// TIA Portal V19 export
FUNCTION "GreiderStyring" : Void   // FC2, LAD
{ S7_Optimized_Access := 'TRUE' }
// stored: SetENOAutomatically false
   VAR_TEMP   // added for the SCL form of the ladder/FBD networks
      _w1 : Bool;
   END_VAR
BEGIN

REGION Network 1
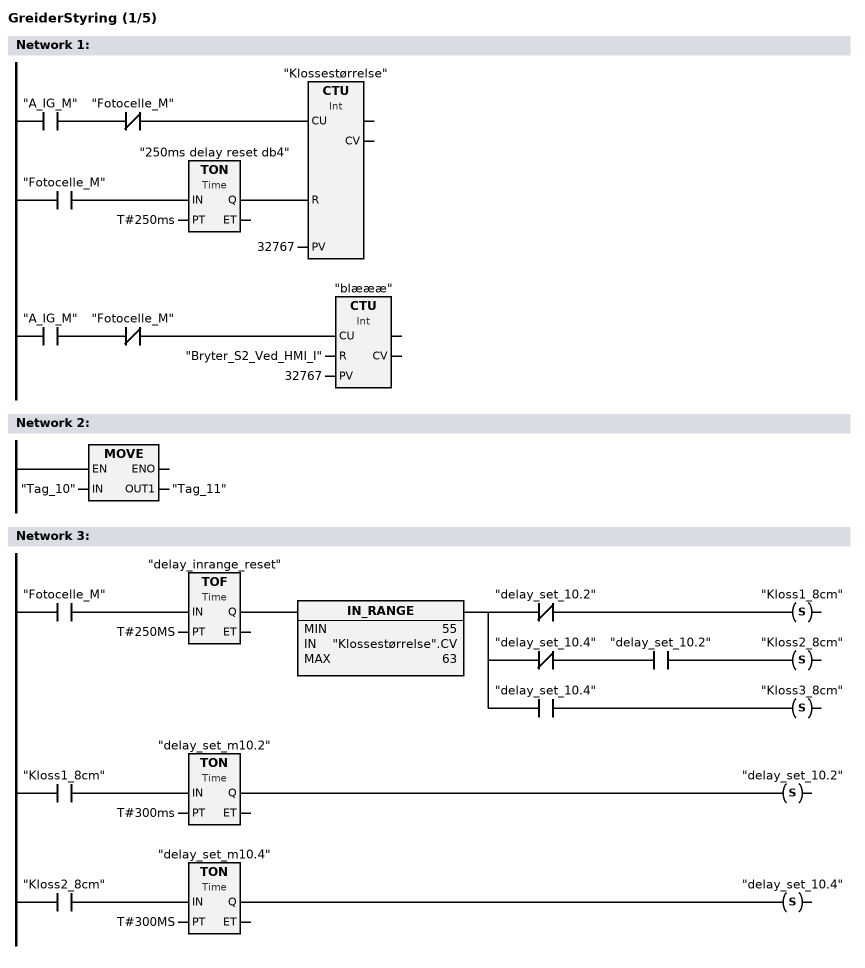
   RUNG wire#powerrail
      Contact( "A_IG_M" )
      I_Contact( "Fotocelle_M" )
      { S7_Templates := "value_type := Int" } "Klossestørrelse".CTU(r := wire#w1, pv := 32767, cv =>)
   END_RUNG
   RUNG wire#powerrail
      Contact( "Fotocelle_M" )
      { S7_Templates := "time_type := Time" } "250ms delay reset db4".TON(pt := T#250ms, et =>)
   END_RUNG wire#w1
   RUNG wire#powerrail
      Contact( "A_IG_M" )
      I_Contact( "Fotocelle_M" )
      { S7_Templates := "value_type := Int" } "blæææ".CTU(r := "Bryter_S2_Ved_HMI_I", pv := 32767, cv =>)
   END_RUNG
   // the same network as SCL:
   "250ms delay reset db4".TON(IN := "Fotocelle_M", PT := T#250ms);
   "Klossestørrelse".CTU(CU := "A_IG_M" AND NOT "Fotocelle_M", R := "250ms delay reset db4".Q, PV := 32767);
   "blæææ".CTU(CU := "A_IG_M" AND NOT "Fotocelle_M", R := "Bryter_S2_Ved_HMI_I", PV := 32767);
END_REGION

REGION Network 2
   RUNG wire#powerrail
      Move(in := "Tag_10", out1 => "Tag_11")
   END_RUNG
   // the same network as SCL:
   "Tag_11" := "Tag_10";
END_REGION

REGION Network 3
   RUNG wire#powerrail
      Contact( "Fotocelle_M" )
      { S7_Templates := "time_type := Time" } "delay_inrange_reset".TOF(pt := T#250MS, et =>)
      { S7_Templates := "SrcType := Int" } InRange(min := 55, in := "Klossestørrelse".CV, max := 63)
      wire#w1
      I_Contact( "delay_set_10.2" )
      S_Coil( "Kloss1_8cm" )
   END_RUNG
   RUNG wire#w1
      I_Contact( "delay_set_10.4" )
      Contact( "delay_set_10.2" )
      S_Coil( "Kloss2_8cm" )
   END_RUNG
   RUNG wire#w1
      Contact( "delay_set_10.4" )
      S_Coil( "Kloss3_8cm" )
   END_RUNG
   RUNG wire#powerrail
      Contact( "Kloss1_8cm" )
      { S7_Templates := "time_type := Time" } "delay_set_m10.2".TON(pt := T#300ms, et =>)
      S_Coil( "delay_set_10.2" )
   END_RUNG
   RUNG wire#powerrail
      Contact( "Kloss2_8cm" )
      { S7_Templates := "time_type := Time" } "delay_set_m10.4".TON(pt := T#300MS, et =>)
      S_Coil( "delay_set_10.4" )
   END_RUNG
   // the same network as SCL:
   "delay_inrange_reset".TOF(IN := "Fotocelle_M", PT := T#250MS);
   #_w1 := "delay_inrange_reset".Q AND (55 <= "Klossestørrelse".CV) AND ("Klossestørrelse".CV <= 63);
   IF #_w1 AND NOT "delay_set_10.2" THEN "Kloss1_8cm" := TRUE; END_IF;
   IF #_w1 AND NOT "delay_set_10.4" AND "delay_set_10.2" THEN "Kloss2_8cm" := TRUE; END_IF;
   IF #_w1 AND "delay_set_10.4" THEN "Kloss3_8cm" := TRUE; END_IF;
   "delay_set_m10.2".TON(IN := "Kloss1_8cm", PT := T#300ms);
   IF "delay_set_m10.2".Q THEN "delay_set_10.2" := TRUE; END_IF;
   "delay_set_m10.4".TON(IN := "Kloss2_8cm", PT := T#300MS);
   IF "delay_set_m10.4".Q THEN "delay_set_10.4" := TRUE; END_IF;
END_REGION

REGION Network 4
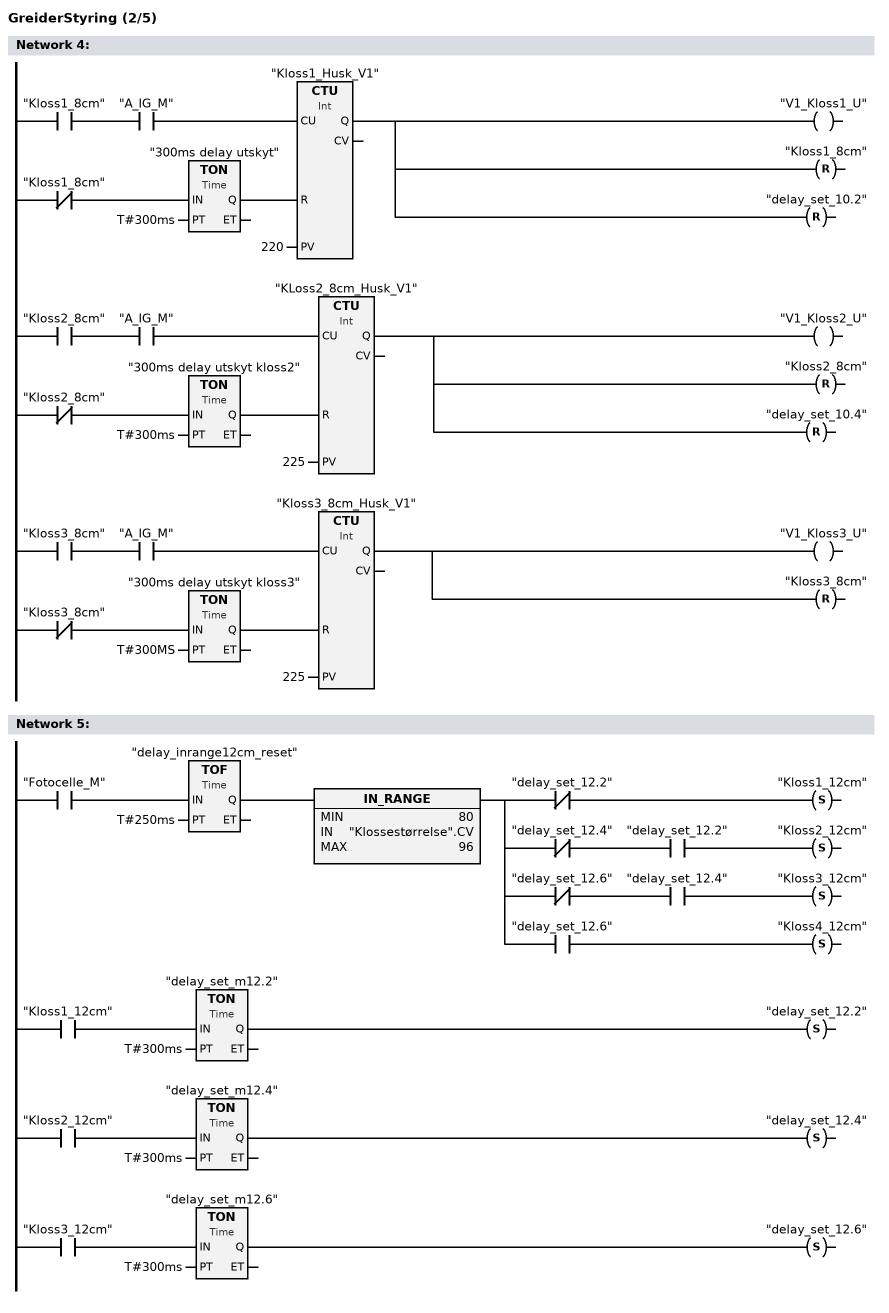
   RUNG wire#powerrail
      Contact( "Kloss1_8cm" )
      Contact( "A_IG_M" )
      { S7_Templates := "value_type := Int" } "Kloss1_Husk_V1".CTU(r := wire#w1, pv := 220, cv =>)
      wire#w2
      Coil( "V1_Kloss1_U" )
   END_RUNG
   RUNG wire#powerrail
      I_Contact( "Kloss1_8cm" )
      { S7_Templates := "time_type := Time" } "300ms delay utskyt".TON(pt := T#300ms, et =>)
   END_RUNG wire#w1
   RUNG wire#w2
      R_Coil( "Kloss1_8cm" )
   END_RUNG
   RUNG wire#w2
      R_Coil( "delay_set_10.2" )
   END_RUNG
   RUNG wire#powerrail
      Contact( "Kloss2_8cm" )
      Contact( "A_IG_M" )
      { S7_Templates := "value_type := Int" } "KLoss2_8cm_Husk_V1".CTU(r := wire#w3, pv := 225, cv =>)
      wire#w4
      Coil( "V1_Kloss2_U" )
   END_RUNG
   RUNG wire#powerrail
      I_Contact( "Kloss2_8cm" )
      { S7_Templates := "time_type := Time" } "300ms delay utskyt kloss2".TON(pt := T#300ms, et =>)
   END_RUNG wire#w3
   RUNG wire#w4
      R_Coil( "Kloss2_8cm" )
   END_RUNG
   RUNG wire#w4
      R_Coil( "delay_set_10.4" )
   END_RUNG
   RUNG wire#powerrail
      Contact( "Kloss3_8cm" )
      Contact( "A_IG_M" )
      { S7_Templates := "value_type := Int" } "Kloss3_8cm_Husk_V1".CTU(r := wire#w5, pv := 225, cv =>)
      wire#w6
      Coil( "V1_Kloss3_U" )
   END_RUNG
   RUNG wire#powerrail
      I_Contact( "Kloss3_8cm" )
      { S7_Templates := "time_type := Time" } "300ms delay utskyt kloss3".TON(pt := T#300MS, et =>)
   END_RUNG wire#w5
   RUNG wire#w6
      R_Coil( "Kloss3_8cm" )
   END_RUNG
   // the same network as SCL:
   "300ms delay utskyt".TON(IN := NOT "Kloss1_8cm", PT := T#300ms);
   "Kloss1_Husk_V1".CTU(CU := "Kloss1_8cm" AND "A_IG_M", R := "300ms delay utskyt".Q, PV := 220);
   "V1_Kloss1_U" := "Kloss1_Husk_V1".Q;
   IF "Kloss1_Husk_V1".Q THEN
       "Kloss1_8cm" := FALSE;
       "delay_set_10.2" := FALSE;
   END_IF;
   "300ms delay utskyt kloss2".TON(IN := NOT "Kloss2_8cm", PT := T#300ms);
   "KLoss2_8cm_Husk_V1".CTU(CU := "Kloss2_8cm" AND "A_IG_M", R := "300ms delay utskyt kloss2".Q, PV := 225);
   "V1_Kloss2_U" := "KLoss2_8cm_Husk_V1".Q;
   IF "KLoss2_8cm_Husk_V1".Q THEN
       "Kloss2_8cm" := FALSE;
       "delay_set_10.4" := FALSE;
   END_IF;
   "300ms delay utskyt kloss3".TON(IN := NOT "Kloss3_8cm", PT := T#300MS);
   "Kloss3_8cm_Husk_V1".CTU(CU := "Kloss3_8cm" AND "A_IG_M", R := "300ms delay utskyt kloss3".Q, PV := 225);
   "V1_Kloss3_U" := "Kloss3_8cm_Husk_V1".Q;
   IF "Kloss3_8cm_Husk_V1".Q THEN "Kloss3_8cm" := FALSE; END_IF;
END_REGION

REGION Network 5
   RUNG wire#powerrail
      Contact( "Fotocelle_M" )
      { S7_Templates := "time_type := Time" } "delay_inrange12cm_reset".TOF(pt := T#250ms, et =>)
      { S7_Templates := "SrcType := Int" } InRange(min := 80, in := "Klossestørrelse".CV, max := 96)
      wire#w1
      I_Contact( "delay_set_12.2" )
      S_Coil( "Kloss1_12cm" )
   END_RUNG
   RUNG wire#w1
      I_Contact( "delay_set_12.4" )
      Contact( "delay_set_12.2" )
      S_Coil( "Kloss2_12cm" )
   END_RUNG
   RUNG wire#w1
      I_Contact( "delay_set_12.6" )
      Contact( "delay_set_12.4" )
      S_Coil( "Kloss3_12cm" )
   END_RUNG
   RUNG wire#w1
      Contact( "delay_set_12.6" )
      S_Coil( "Kloss4_12cm" )
   END_RUNG
   RUNG wire#powerrail
      Contact( "Kloss1_12cm" )
      { S7_Templates := "time_type := Time" } "delay_set_m12.2".TON(pt := T#300ms, et =>)
      S_Coil( "delay_set_12.2" )
   END_RUNG
   RUNG wire#powerrail
      Contact( "Kloss2_12cm" )
      { S7_Templates := "time_type := Time" } "delay_set_m12.4".TON(pt := T#300ms, et =>)
      S_Coil( "delay_set_12.4" )
   END_RUNG
   RUNG wire#powerrail
      Contact( "Kloss3_12cm" )
      { S7_Templates := "time_type := Time" } "delay_set_m12.6".TON(pt := T#300ms, et =>)
      S_Coil( "delay_set_12.6" )
   END_RUNG
   // the same network as SCL:
   "delay_inrange12cm_reset".TOF(IN := "Fotocelle_M", PT := T#250ms);
   #_w1 := "delay_inrange12cm_reset".Q AND (80 <= "Klossestørrelse".CV) AND ("Klossestørrelse".CV <= 96);
   IF #_w1 AND NOT "delay_set_12.2" THEN "Kloss1_12cm" := TRUE; END_IF;
   IF #_w1 AND NOT "delay_set_12.4" AND "delay_set_12.2" THEN "Kloss2_12cm" := TRUE; END_IF;
   IF #_w1 AND NOT "delay_set_12.6" AND "delay_set_12.4" THEN "Kloss3_12cm" := TRUE; END_IF;
   IF #_w1 AND "delay_set_12.6" THEN "Kloss4_12cm" := TRUE; END_IF;
   "delay_set_m12.2".TON(IN := "Kloss1_12cm", PT := T#300ms);
   IF "delay_set_m12.2".Q THEN "delay_set_12.2" := TRUE; END_IF;
   "delay_set_m12.4".TON(IN := "Kloss2_12cm", PT := T#300ms);
   IF "delay_set_m12.4".Q THEN "delay_set_12.4" := TRUE; END_IF;
   "delay_set_m12.6".TON(IN := "Kloss3_12cm", PT := T#300ms);
   IF "delay_set_m12.6".Q THEN "delay_set_12.6" := TRUE; END_IF;
END_REGION

REGION Network 6
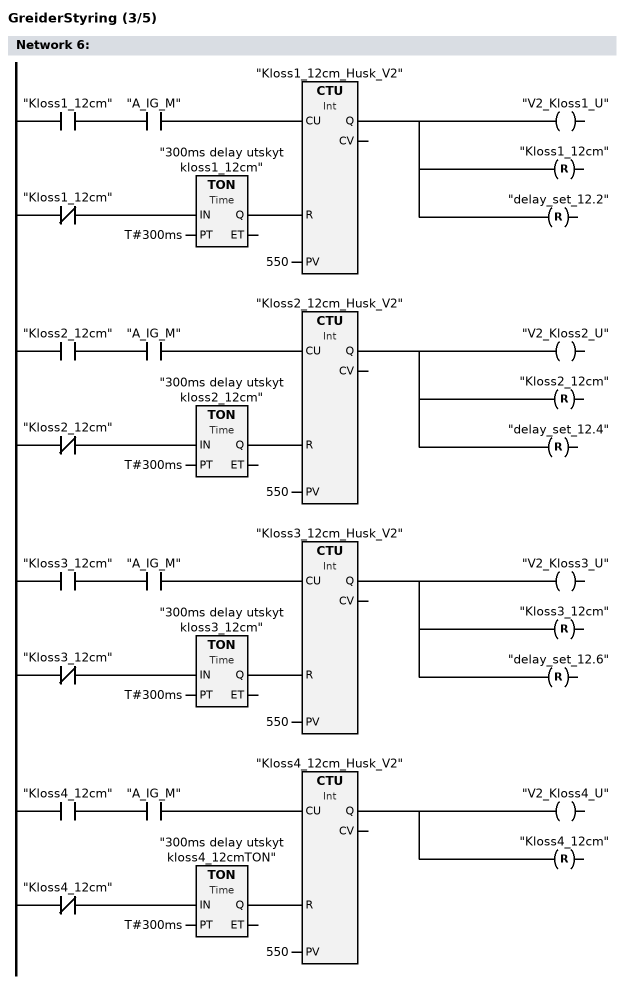
   RUNG wire#powerrail
      Contact( "Kloss1_12cm" )
      Contact( "A_IG_M" )
      { S7_Templates := "value_type := Int" } "Kloss1_12cm_Husk_V2".CTU(r := wire#w1, pv := 550, cv =>)
      wire#w2
      Coil( "V2_Kloss1_U" )
   END_RUNG
   RUNG wire#powerrail
      I_Contact( "Kloss1_12cm" )
      { S7_Templates := "time_type := Time" } "300ms delay utskyt kloss1_12cm".TON(pt := T#300ms, et =>)
   END_RUNG wire#w1
   RUNG wire#w2
      R_Coil( "Kloss1_12cm" )
   END_RUNG
   RUNG wire#w2
      R_Coil( "delay_set_12.2" )
   END_RUNG
   RUNG wire#powerrail
      Contact( "Kloss2_12cm" )
      Contact( "A_IG_M" )
      { S7_Templates := "value_type := Int" } "Kloss2_12cm_Husk_V2".CTU(r := wire#w3, pv := 550, cv =>)
      wire#w4
      Coil( "V2_Kloss2_U" )
   END_RUNG
   RUNG wire#powerrail
      I_Contact( "Kloss2_12cm" )
      { S7_Templates := "time_type := Time" } "300ms delay utskyt kloss2_12cm".TON(pt := T#300ms, et =>)
   END_RUNG wire#w3
   RUNG wire#w4
      R_Coil( "Kloss2_12cm" )
   END_RUNG
   RUNG wire#w4
      R_Coil( "delay_set_12.4" )
   END_RUNG
   RUNG wire#powerrail
      Contact( "Kloss3_12cm" )
      Contact( "A_IG_M" )
      { S7_Templates := "value_type := Int" } "Kloss3_12cm_Husk_V2".CTU(r := wire#w5, pv := 550, cv =>)
      wire#w6
      Coil( "V2_Kloss3_U" )
   END_RUNG
   RUNG wire#powerrail
      I_Contact( "Kloss3_12cm" )
      { S7_Templates := "time_type := Time" } "300ms delay utskyt kloss3_12cm".TON(pt := T#300ms, et =>)
   END_RUNG wire#w5
   RUNG wire#w6
      R_Coil( "Kloss3_12cm" )
   END_RUNG
   RUNG wire#w6
      R_Coil( "delay_set_12.6" )
   END_RUNG
   RUNG wire#powerrail
      Contact( "Kloss4_12cm" )
      Contact( "A_IG_M" )
      { S7_Templates := "value_type := Int" } "Kloss4_12cm_Husk_V2".CTU(r := wire#w7, pv := 550, cv =>)
      wire#w8
      Coil( "V2_Kloss4_U" )
   END_RUNG
   RUNG wire#powerrail
      I_Contact( "Kloss4_12cm" )
      { S7_Templates := "time_type := Time" } "300ms delay utskyt kloss4_12cmTON".TON(pt := T#300ms, et =>)
   END_RUNG wire#w7
   RUNG wire#w8
      R_Coil( "Kloss4_12cm" )
   END_RUNG
   // the same network as SCL:
   "300ms delay utskyt kloss1_12cm".TON(IN := NOT "Kloss1_12cm", PT := T#300ms);
   "Kloss1_12cm_Husk_V2".CTU(CU := "Kloss1_12cm" AND "A_IG_M",
                           R := "300ms delay utskyt kloss1_12cm".Q,
                           PV := 550);
   "V2_Kloss1_U" := "Kloss1_12cm_Husk_V2".Q;
   IF "Kloss1_12cm_Husk_V2".Q THEN
       "Kloss1_12cm" := FALSE;
       "delay_set_12.2" := FALSE;
   END_IF;
   "300ms delay utskyt kloss2_12cm".TON(IN := NOT "Kloss2_12cm", PT := T#300ms);
   "Kloss2_12cm_Husk_V2".CTU(CU := "Kloss2_12cm" AND "A_IG_M",
                           R := "300ms delay utskyt kloss2_12cm".Q,
                           PV := 550);
   "V2_Kloss2_U" := "Kloss2_12cm_Husk_V2".Q;
   IF "Kloss2_12cm_Husk_V2".Q THEN
       "Kloss2_12cm" := FALSE;
       "delay_set_12.4" := FALSE;
   END_IF;
   "300ms delay utskyt kloss3_12cm".TON(IN := NOT "Kloss3_12cm", PT := T#300ms);
   "Kloss3_12cm_Husk_V2".CTU(CU := "Kloss3_12cm" AND "A_IG_M",
                           R := "300ms delay utskyt kloss3_12cm".Q,
                           PV := 550);
   "V2_Kloss3_U" := "Kloss3_12cm_Husk_V2".Q;
   IF "Kloss3_12cm_Husk_V2".Q THEN
       "Kloss3_12cm" := FALSE;
       "delay_set_12.6" := FALSE;
   END_IF;
   "300ms delay utskyt kloss4_12cmTON".TON(IN := NOT "Kloss4_12cm", PT := T#300ms);
   "Kloss4_12cm_Husk_V2".CTU(CU := "Kloss4_12cm" AND "A_IG_M",
                           R := "300ms delay utskyt kloss4_12cmTON".Q,
                           PV := 550);
   "V2_Kloss4_U" := "Kloss4_12cm_Husk_V2".Q;
   IF "Kloss4_12cm_Husk_V2".Q THEN "Kloss4_12cm" := FALSE; END_IF;
END_REGION

REGION Network 7
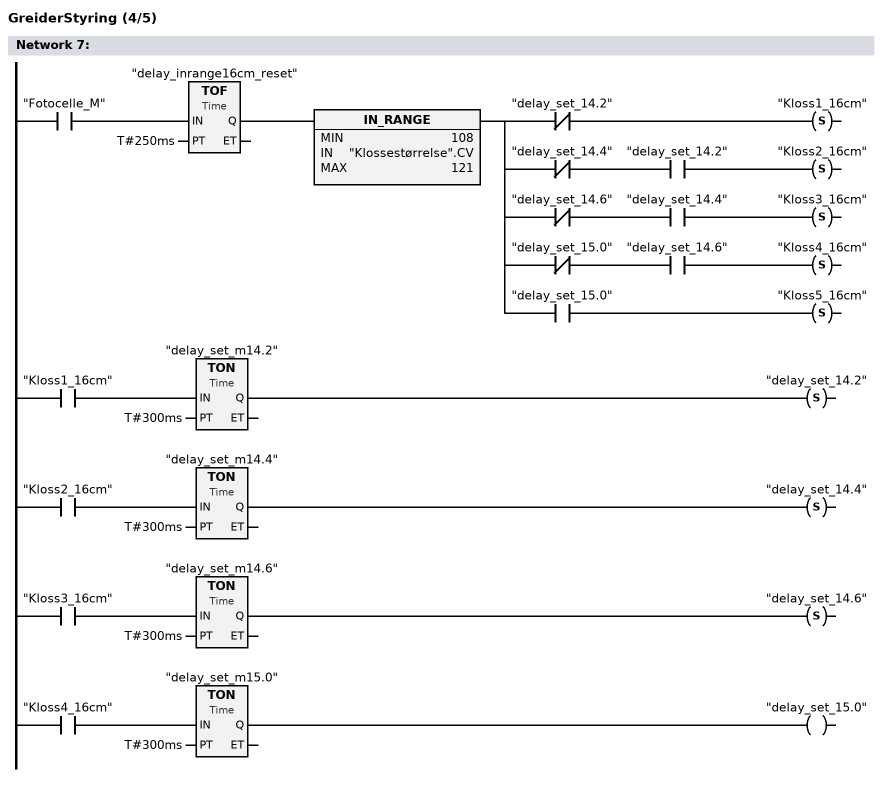
   RUNG wire#powerrail
      Contact( "Fotocelle_M" )
      { S7_Templates := "time_type := Time" } "delay_inrange16cm_reset".TOF(pt := T#250ms, et =>)
      { S7_Templates := "SrcType := Int" } InRange(min := 108, in := "Klossestørrelse".CV, max := 121)
      wire#w1
      I_Contact( "delay_set_14.2" )
      S_Coil( "Kloss1_16cm" )
   END_RUNG
   RUNG wire#w1
      I_Contact( "delay_set_14.4" )
      Contact( "delay_set_14.2" )
      S_Coil( "Kloss2_16cm" )
   END_RUNG
   RUNG wire#w1
      I_Contact( "delay_set_14.6" )
      Contact( "delay_set_14.4" )
      S_Coil( "Kloss3_16cm" )
   END_RUNG
   RUNG wire#w1
      I_Contact( "delay_set_15.0" )
      Contact( "delay_set_14.6" )
      S_Coil( "Kloss4_16cm" )
   END_RUNG
   RUNG wire#w1
      Contact( "delay_set_15.0" )
      S_Coil( "Kloss5_16cm" )
   END_RUNG
   RUNG wire#powerrail
      Contact( "Kloss1_16cm" )
      { S7_Templates := "time_type := Time" } "delay_set_m14.2".TON(pt := T#300ms, et =>)
      S_Coil( "delay_set_14.2" )
   END_RUNG
   RUNG wire#powerrail
      Contact( "Kloss2_16cm" )
      { S7_Templates := "time_type := Time" } "delay_set_m14.4".TON(pt := T#300ms, et =>)
      S_Coil( "delay_set_14.4" )
   END_RUNG
   RUNG wire#powerrail
      Contact( "Kloss3_16cm" )
      { S7_Templates := "time_type := Time" } "delay_set_m14.6".TON(pt := T#300ms, et =>)
      S_Coil( "delay_set_14.6" )
   END_RUNG
   RUNG wire#powerrail
      Contact( "Kloss4_16cm" )
      { S7_Templates := "time_type := Time" } "delay_set_m15.0".TON(pt := T#300ms, et =>)
      Coil( "delay_set_15.0" )
   END_RUNG
   // the same network as SCL:
   "delay_inrange16cm_reset".TOF(IN := "Fotocelle_M", PT := T#250ms);
   #_w1 := "delay_inrange16cm_reset".Q AND (108 <= "Klossestørrelse".CV) AND ("Klossestørrelse".CV <= 121);
   IF #_w1 AND NOT "delay_set_14.2" THEN "Kloss1_16cm" := TRUE; END_IF;
   IF #_w1 AND NOT "delay_set_14.4" AND "delay_set_14.2" THEN "Kloss2_16cm" := TRUE; END_IF;
   IF #_w1 AND NOT "delay_set_14.6" AND "delay_set_14.4" THEN "Kloss3_16cm" := TRUE; END_IF;
   IF #_w1 AND NOT "delay_set_15.0" AND "delay_set_14.6" THEN "Kloss4_16cm" := TRUE; END_IF;
   IF #_w1 AND "delay_set_15.0" THEN "Kloss5_16cm" := TRUE; END_IF;
   "delay_set_m14.2".TON(IN := "Kloss1_16cm", PT := T#300ms);
   IF "delay_set_m14.2".Q THEN "delay_set_14.2" := TRUE; END_IF;
   "delay_set_m14.4".TON(IN := "Kloss2_16cm", PT := T#300ms);
   IF "delay_set_m14.4".Q THEN "delay_set_14.4" := TRUE; END_IF;
   "delay_set_m14.6".TON(IN := "Kloss3_16cm", PT := T#300ms);
   IF "delay_set_m14.6".Q THEN "delay_set_14.6" := TRUE; END_IF;
   "delay_set_m15.0".TON(IN := "Kloss4_16cm", PT := T#300ms);
   "delay_set_15.0" := "delay_set_m15.0".Q;
END_REGION

REGION Network 8
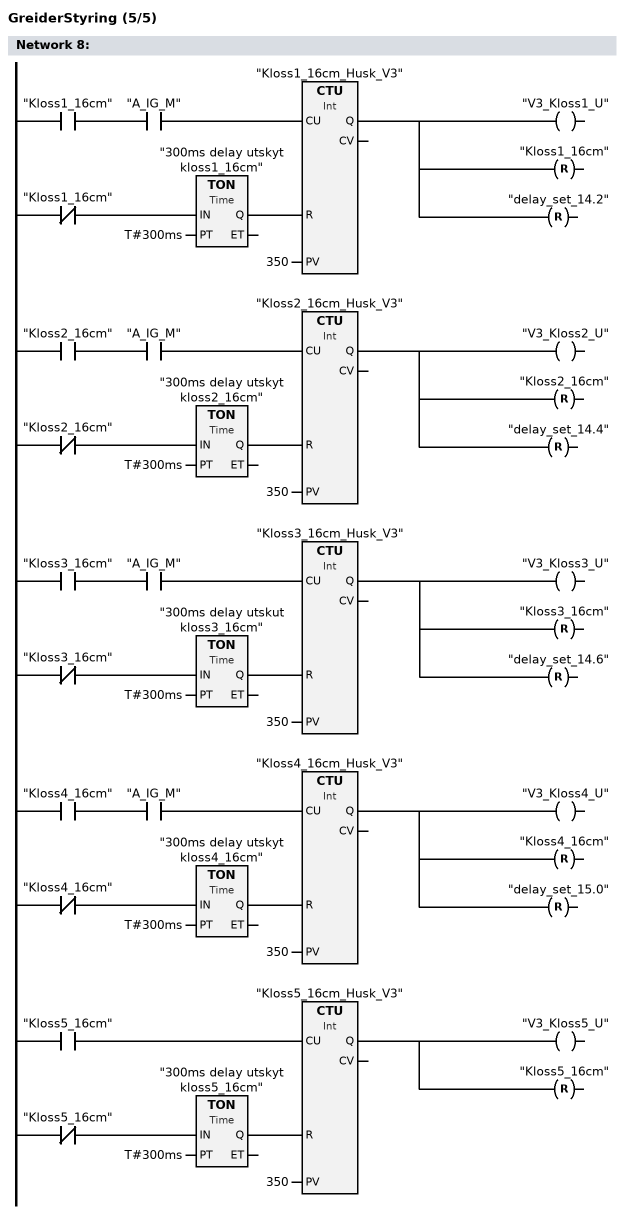
   RUNG wire#powerrail
      Contact( "Kloss1_16cm" )
      Contact( "A_IG_M" )
      { S7_Templates := "value_type := Int" } "Kloss1_16cm_Husk_V3".CTU(r := wire#w1, pv := 350, cv =>)
      wire#w2
      Coil( "V3_Kloss1_U" )
   END_RUNG
   RUNG wire#powerrail
      I_Contact( "Kloss1_16cm" )
      { S7_Templates := "time_type := Time" } "300ms delay utskyt kloss1_16cm".TON(pt := T#300ms, et =>)
   END_RUNG wire#w1
   RUNG wire#w2
      R_Coil( "Kloss1_16cm" )
   END_RUNG
   RUNG wire#w2
      R_Coil( "delay_set_14.2" )
   END_RUNG
   RUNG wire#powerrail
      Contact( "Kloss2_16cm" )
      Contact( "A_IG_M" )
      { S7_Templates := "value_type := Int" } "Kloss2_16cm_Husk_V3".CTU(r := wire#w3, pv := 350, cv =>)
      wire#w4
      Coil( "V3_Kloss2_U" )
   END_RUNG
   RUNG wire#powerrail
      I_Contact( "Kloss2_16cm" )
      { S7_Templates := "time_type := Time" } "300ms delay utskyt kloss2_16cm".TON(pt := T#300ms, et =>)
   END_RUNG wire#w3
   RUNG wire#w4
      R_Coil( "Kloss2_16cm" )
   END_RUNG
   RUNG wire#w4
      R_Coil( "delay_set_14.4" )
   END_RUNG
   RUNG wire#powerrail
      Contact( "Kloss3_16cm" )
      Contact( "A_IG_M" )
      { S7_Templates := "value_type := Int" } "Kloss3_16cm_Husk_V3".CTU(r := wire#w5, pv := 350, cv =>)
      wire#w6
      Coil( "V3_Kloss3_U" )
   END_RUNG
   RUNG wire#powerrail
      I_Contact( "Kloss3_16cm" )
      { S7_Templates := "time_type := Time" } "300ms delay utskut kloss3_16cm".TON(pt := T#300ms, et =>)
   END_RUNG wire#w5
   RUNG wire#w6
      R_Coil( "Kloss3_16cm" )
   END_RUNG
   RUNG wire#w6
      R_Coil( "delay_set_14.6" )
   END_RUNG
   RUNG wire#powerrail
      Contact( "Kloss4_16cm" )
      Contact( "A_IG_M" )
      { S7_Templates := "value_type := Int" } "Kloss4_16cm_Husk_V3".CTU(r := wire#w7, pv := 350, cv =>)
      wire#w8
      Coil( "V3_Kloss4_U" )
   END_RUNG
   RUNG wire#powerrail
      I_Contact( "Kloss4_16cm" )
      { S7_Templates := "time_type := Time" } "300ms delay utskyt kloss4_16cm".TON(pt := T#300ms, et =>)
   END_RUNG wire#w7
   RUNG wire#w8
      R_Coil( "Kloss4_16cm" )
   END_RUNG
   RUNG wire#w8
      R_Coil( "delay_set_15.0" )
   END_RUNG
   RUNG wire#powerrail
      Contact( "Kloss5_16cm" )
      { S7_Templates := "value_type := Int" } "Kloss5_16cm_Husk_V3".CTU(r := wire#w9, pv := 350, cv =>)
      wire#w10
      Coil( "V3_Kloss5_U" )
   END_RUNG
   RUNG wire#powerrail
      I_Contact( "Kloss5_16cm" )
      { S7_Templates := "time_type := Time" } "300ms delay utskyt kloss5_16cm".TON(pt := T#300ms, et =>)
   END_RUNG wire#w9
   RUNG wire#w10
      R_Coil( "Kloss5_16cm" )
   END_RUNG
   // the same network as SCL:
   "300ms delay utskyt kloss1_16cm".TON(IN := NOT "Kloss1_16cm", PT := T#300ms);
   "Kloss1_16cm_Husk_V3".CTU(CU := "Kloss1_16cm" AND "A_IG_M",
                           R := "300ms delay utskyt kloss1_16cm".Q,
                           PV := 350);
   "V3_Kloss1_U" := "Kloss1_16cm_Husk_V3".Q;
   IF "Kloss1_16cm_Husk_V3".Q THEN
       "Kloss1_16cm" := FALSE;
       "delay_set_14.2" := FALSE;
   END_IF;
   "300ms delay utskyt kloss2_16cm".TON(IN := NOT "Kloss2_16cm", PT := T#300ms);
   "Kloss2_16cm_Husk_V3".CTU(CU := "Kloss2_16cm" AND "A_IG_M",
                           R := "300ms delay utskyt kloss2_16cm".Q,
                           PV := 350);
   "V3_Kloss2_U" := "Kloss2_16cm_Husk_V3".Q;
   IF "Kloss2_16cm_Husk_V3".Q THEN
       "Kloss2_16cm" := FALSE;
       "delay_set_14.4" := FALSE;
   END_IF;
   "300ms delay utskut kloss3_16cm".TON(IN := NOT "Kloss3_16cm", PT := T#300ms);
   "Kloss3_16cm_Husk_V3".CTU(CU := "Kloss3_16cm" AND "A_IG_M",
                           R := "300ms delay utskut kloss3_16cm".Q,
                           PV := 350);
   "V3_Kloss3_U" := "Kloss3_16cm_Husk_V3".Q;
   IF "Kloss3_16cm_Husk_V3".Q THEN
       "Kloss3_16cm" := FALSE;
       "delay_set_14.6" := FALSE;
   END_IF;
   "300ms delay utskyt kloss4_16cm".TON(IN := NOT "Kloss4_16cm", PT := T#300ms);
   "Kloss4_16cm_Husk_V3".CTU(CU := "Kloss4_16cm" AND "A_IG_M",
                           R := "300ms delay utskyt kloss4_16cm".Q,
                           PV := 350);
   "V3_Kloss4_U" := "Kloss4_16cm_Husk_V3".Q;
   IF "Kloss4_16cm_Husk_V3".Q THEN
       "Kloss4_16cm" := FALSE;
       "delay_set_15.0" := FALSE;
   END_IF;
   "300ms delay utskyt kloss5_16cm".TON(IN := NOT "Kloss5_16cm", PT := T#300ms);
   "Kloss5_16cm_Husk_V3".CTU(CU := "Kloss5_16cm", R := "300ms delay utskyt kloss5_16cm".Q, PV := 350);
   "V3_Kloss5_U" := "Kloss5_16cm_Husk_V3".Q;
   IF "Kloss5_16cm_Husk_V3".Q THEN "Kloss5_16cm" := FALSE; END_IF;
END_REGION
END_FUNCTION
